Yaskawa INFORM job: B-2-08279-80-SUB-M.JBI

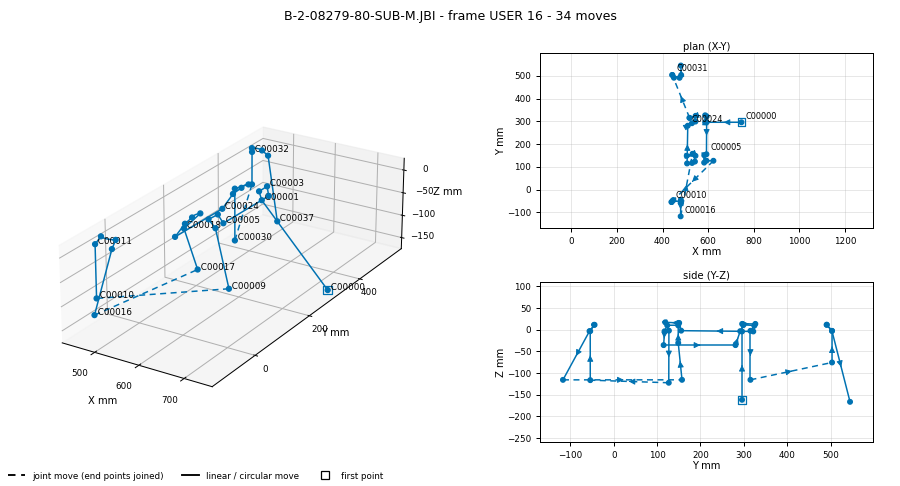
[picture p0: tool path of B-2-08279-80-SUB-M.JBI in frame USER 16, 34 of 38 moves have a stored position in this frame; points joined in program order, loops and branches not executed]
/JOB
//NAME B-2-08279-80-SUB-M
///FOLDERNAME PART_420-08279-80
//POS
///NPOS 38,0,38,0,0,0
///USER 16
///TOOL 4
///POSTYPE USER
///RECTAN
///RCONF 1,0,0,0,0,0,0,0,0,0,0,0,0,0,0,0,0,0,0,0,0,0,0,0
C00000=746.323,295.750,-161.584,-27.8970,11.3047,78.2347
C00001=593.519,295.721,-3.979,-46.5250,6.9320,75.2540
C00002=587.014,296.060,13.448,-46.5201,6.9370,75.2616
C00003=587.012,326.450,13.446,-46.5198,6.9375,75.2618
C00004=593.755,321.720,-3.979,-46.5250,6.9320,75.2540
C00005=592.773,155.478,-2.185,-42.9430,-21.0870,89.6170
C00006=583.161,150.868,15.675,-42.9431,-21.0924,89.6126
C00007=582.722,118.727,17.083,-42.9400,-21.0914,89.6135
C00008=592.773,127.194,-2.185,-42.9430,-21.0870,89.6170
C00009=623.287,126.871,-122.266,-42.9430,-21.0870,89.6170
C00010=439.578,-54.115,-116.298,-6.5594,-44.9787,-116.9695
C00011=439.802,-54.182,-3.282,-6.5590,-44.9790,-116.9690
C00012=447.518,-45.323,11.359,-6.5584,-44.9789,-116.9674
C00013=460.761,-50.523,12.098,-6.5566,-44.9776,-90.5193
C00014=480.522,-44.190,11.330,-6.5534,-44.9795,-55.2571
C00015=479.608,-55.834,-3.282,-6.5580,-44.9790,-55.2560
C00016=479.541,-117.038,-115.581,-6.5567,-44.9793,-55.2560
C00017=531.608,157.384,-115.500,-16.3490,-44.1220,152.7880
C00018=506.244,148.712,-30.487,-12.7418,-45.3534,179.0535
C00019=544.617,148.640,9.985,-12.7408,-45.3527,179.0534
C00020=540.216,134.630,10.365,-17.0917,-44.8745,-157.0797
C00021=542.140,123.298,10.114,-16.5146,-44.7717,-145.3138
C00022=529.621,117.175,-3.669,-16.5140,-44.7720,-151.5720
C00023=507.748,115.031,-35.500,-16.5140,-44.7720,-151.5720
C00024=510.771,280.690,-35.500,3.4420,-44.9790,-154.0720
C00025=529.020,291.566,-3.353,3.4420,-44.9790,-154.0720
C00026=544.383,298.817,10.706,3.4420,-44.9788,-154.0716
C00027=542.128,309.287,10.661,7.8953,-43.2349,176.8662
C00028=545.226,324.093,9.237,15.6705,-44.9799,144.2120
C00029=518.589,315.156,-2.528,16.5470,-44.9790,144.2150
C00030=518.589,315.156,-115.500,16.5470,-44.9790,144.2150
C00031=442.808,503.260,-75.500,28.9260,-36.2220,77.7090
C00032=442.809,503.258,-2.647,28.9260,-36.2220,77.7090
C00033=450.033,491.127,11.426,28.9260,-36.2221,77.7084
C00034=461.340,495.208,11.490,15.7357,-42.8114,71.8249
C00035=474.608,490.859,11.478,13.1197,-43.5301,40.3824
C00036=481.884,503.018,-2.647,12.3290,-43.7170,41.5290
C00037=480.362,544.738,-166.231,12.0346,-43.7826,41.9531
///TOOL 0
///POSTYPE ANGLE
///ANGLE
EC00000=-45.0000
///TOOL 4
EC00001=-45.0000
///TOOL 0
EC00002=-45.0000
EC00003=-45.0000
///TOOL 4
EC00004=-45.0000
EC00005=-45.0000
///TOOL 0
EC00006=-45.0005
EC00007=-45.0005
///TOOL 4
EC00008=-45.0000
EC00009=-45.0000
///TOOL 0
EC00010=-90.0000
///TOOL 4
EC00011=-90.0000
///TOOL 0
EC00012=-90.0000
EC00013=-90.0000
EC00014=-90.0000
///TOOL 4
EC00015=-90.0000
///TOOL 0
EC00016=-90.0000
///TOOL 4
EC00017=-90.0000
///TOOL 0
EC00018=-90.0000
EC00019=-90.0000
EC00020=-90.0000
EC00021=-90.0000
///TOOL 4
EC00022=-90.0000
EC00023=-90.0000
EC00024=-90.0000
EC00025=-90.0000
///TOOL 0
EC00026=-90.0000
EC00027=-90.0000
EC00028=-90.0000
///TOOL 4
EC00029=-90.0000
EC00030=-90.0000
EC00031=-90.0000
EC00032=-90.0000
///TOOL 0
EC00033=-90.0000
EC00034=-90.0000
EC00035=-90.0000
///TOOL 4
EC00036=-90.0000
///TOOL 0
EC00037=-90.0000
//INST
///DATE 2021/10/29 11:36
///ATTR SC,RW,RJ
////FRAME USER 16
///GROUP1 RB1
///GROUP2 ST3
NOP
'Path Start: PP9
'Warning, the first motion progra
'mmed for this routine was not a
'joint motion
'The following movement has been
'added. Please update your OCTOPU
'Z simulation.
MOVJ C00000 VJ=100.00  +MOVJ EC00000
SMOVL C00001 V=1250.0  +MOVJ EC00001
SMOVL C00002 V=300.0  +MOVJ EC00002
ARCON ASF#(951)
SMOVL C00003 V=8.5  +MOVJ EC00003
ARCOF AEF#(951)
SMOVL C00004 V=1250.0  +MOVJ EC00004
'Path End
'Path Start: PP15
SMOVL C00005 V=1250.0  +MOVJ EC00005
SMOVL C00006 V=300.0  +MOVJ EC00006
ARCON ASF#(951)
SMOVL C00007  +MOVJ EC00007
ARCOF AEF#(951)
SMOVL C00008 V=1250.0  +MOVJ EC00008
SMOVL C00009 V=1250.0  +MOVJ EC00009
'Path End
'Path Start: PP16
MOVJ C00010 VJ=25.00  +MOVJ EC00010
SMOVL C00011 V=1250.0  +MOVJ EC00011
SMOVC C00012 V=300.0  +MOVJ EC00012
ARCON ASF#(951)
SMOVC C00013 V=8.5  +MOVJ EC00013
SMOVC C00014 V=8.5  +MOVJ EC00014
ARCOF AEF#(951)
SMOVL C00015 V=1250.0  +MOVJ EC00015
SMOVL C00016 V=1250.0  +MOVJ EC00016
'Path End
'Path Start: PP19
MOVJ C00017 VJ=100.00  +MOVJ EC00017
SMOVL C00018 V=1250.0  +MOVJ EC00018
SMOVC C00019 V=300.0  +MOVJ EC00019
ARCON ASF#(951)
SMOVC C00020 V=8.5  +MOVJ EC00020
SMOVC C00021 V=8.5  +MOVJ EC00021
ARCOF AEF#(951)
SMOVL C00022 V=1250.0  +MOVJ EC00022
SMOVL C00023 V=1250.0  +MOVJ EC00023
'Path End
'Path Start: PP20
SMOVL C00024 V=1250.0  +MOVJ EC00024
SMOVL C00025 V=1250.0  +MOVJ EC00025
SMOVC C00026 V=300.0  +MOVJ EC00026
ARCON ASF#(951)
SMOVC C00027 V=8.5  +MOVJ EC00027
SMOVC C00028 V=8.5  +MOVJ EC00028
ARCOF AEF#(951)
SMOVL C00029 V=1250.0  +MOVJ EC00029
SMOVL C00030 V=1250.0  +MOVJ EC00030
'Path End
'Path Start: PP22
MOVJ C00031 VJ=100.00  +MOVJ EC00031
SMOVL C00032 V=1250.0  +MOVJ EC00032
SMOVC C00033 V=300.0  +MOVJ EC00033
ARCON ASF#(951)
SMOVC C00034 V=8.5  +MOVJ EC00034
SMOVC C00035 V=8.5  +MOVJ EC00035
ARCOF AEF#(951)
SMOVL C00036 V=1250.0  +MOVJ EC00036
SMOVL C00037 V=1250.0  +MOVJ EC00037
'Path End
END
